Staubli VAL3: convSelect.pgx

program convSelect(string& x_sFileName[] (dimensions=1), num& x_nError[] (dimensions=1), bool& x_bQuit[] (dimensions=1))
  local bool l_bIsInList
  local bool l_bQuit
  local bool l_bRefresh
  local num l_nError
  local num l_nIdx
  local num l_nKeyPressed
  local string l_sEmpty
  local string l_sFileName
  local string l_sNewFileName
begin
  // This program allows the user to select a conveyor calibration
  // file from a list or to enter a new calibration filename.
  // The selected file is loaded into the memory
  //
  //----------------------------------------------------------------
  //
  //**************************
  //***** INITALIZATIONS *****
  //**************************
  l_bQuit=false
  l_nError=-1
  l_bRefresh=true
  x_nError=0
  x_bQuit=false
  libList(cfg:sPATHCONVEYOR,sItemList)
  l_sEmpty=""
  //
  //**************************
  //***** EVENT SECTION  *****
  //**************************
  do
    // Display page and list existing conveyor libraries
    call lang:Page(60,l_sEmpty,sel(len(sItemList[0])!=0,10,11),l_bRefresh,l_nKeyPressed)
    if l_bRefresh==true
      call _displayList(cfg:sPATHCONVEYOR,lang:sListOfMessage[9],22,2,15,7)
      l_bRefresh=false
    endIf
    //
    call up:listEvent(l_nKeyPressed,l_nIdx,l_sFileName)
    switch l_nKeyPressed
      // New
      case 2
        call convGetName(l_sNewFileName)
        l_sFileName=l_sNewFileName
        // Check file name
        if len(l_sFileName)!=0
          call isInList(l_sFileName,sItemList,l_bIsInList)
          if !l_bIsInList
            // Load conveyor template
            l_nError=cnv:libLoad(cfg:sPATHTEMPLATE+cfg:sGENERICCONV)
            // Select Encoder Lib,Detection Lib etc...
            call convConfig(l_nError)
            switch l_nError
              // All right
              case 0
                // Create conveyor
                call convCreate(l_sFileName,l_nError)
                if l_nError==0
                  call convLoad(l_sFileName,l_nError)
                  if l_nError==0
                    x_sFileName=l_sFileName
                  endIf
                else
                  x_nError=l_nError
                endIf
                l_bQuit=true
              break
              case -1
                // Operation canceled by user
                l_bRefresh=true
              break
              default
                //call up:msgBox(sErrorMessage,36,lang:sMenu[1],l_nKeyPressed)
                x_nError=l_nError
                l_bQuit=true
              break
            endSwitch
          endIf
        else
          l_bRefresh=true
        endIf
      break
      // Duplicate
      case 3
        call convLoad(l_sFileName,l_nError)
        if l_nError==0
          // display library list again
          call lang:Page(60,l_sEmpty,sel(len(sItemList[0])!=0,10,11),true,l_nKeyPressed)
          call _displayList(cfg:sPATHCONVEYOR,lang:sListOfMessage[9],22,2,15,7)
          call convGetName(l_sNewFileName)
          l_sFileName=l_sNewFileName
          if len(l_sFileName)!=0
            call convCreate(l_sFileName,l_nError)
            if l_nError!=0
              call up:msgBox(lang:sListOfMessage[36],36,lang:sMenu[1],l_nKeyPressed)
            endIf
          endIf
        else
          l_bQuit=true
          x_nError=l_nError
        endIf
        l_bRefresh=true
      break
      // Select or Return
      case 4,270
        call convLoad(l_sFileName,x_nError)
        if x_nError==0
          x_sFileName=l_sFileName
        else
        endIf
        l_bQuit=true
      break
      // Delete
      case 6
        call ut:addStrToString(lang:sListOfMessage[16],sErrorMessage,"",l_sFileName)
        call up:msgBox(sErrorMessage,36,lang:sMenu[21],l_nKeyPressed)
        if l_nKeyPressed==3
          // Answer is Yes
          l_nError=libDelete(cfg:sPATHCONVEYOR+l_sFileName)
          libList(cfg:sPATHCONVEYOR,sItemList)
        else
        endIf
        l_bRefresh=true
      break
      // Cancel
      case 8
        l_bQuit=true
        x_bQuit=true
      break
    endSwitch
    delay(0)
  until (l_bQuit==true)
  cls()
end
